// TIA Portal V19 export
FUNCTION "AFC_Steptimer" : Void   // FC35, FBD
TITLE = AFC_Steptimer
{ S7_Optimized_Access := 'TRUE' }
AUTHOR : CH
FAMILY : Aktina
NAME : Global
// AFC_Steptimer
// stored: AutoNumber false, SetENOAutomatically false
   VAR_INPUT
      "step" : Bool;   // Step activated
      count_max : Bool;   // Trigger for max step timer
      count_step : Bool;   // Trigger for conditional step timer
      Pulse : Bool;   // Pulse used for time count
      reset_max : Bool;   // Reset max step timer
      reset_step : Bool;   // Reset conditional step timer
      reset_warn : Bool;   // Reset max timer warning
   END_VAR
   VAR_OUTPUT
      max_warn : Bool;   // Max step timer has elapsed
   END_VAR
   VAR_IN_OUT
      Data : Variant;   // Unique data area for this counter
   END_VAR
   VAR_TEMP
      i : "UDT_STEPTIMER";
      logical1 : Bool;
      remain : UDInt;
      intermediate : UDInt;
      sec : UDInt;
      min : UDInt;
      hour : UDInt;
   END_VAR
BEGIN

REGION Network 1: GEN: Create Logical 1
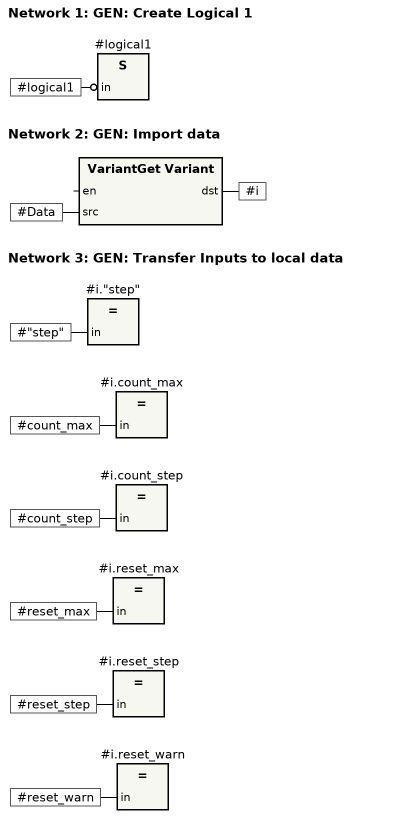
   IF NOT #logical1 THEN #logical1 := TRUE; END_IF;
END_REGION

REGION Network 2: GEN: Import data
   // no SCL statement known for VariantGet: written as a call
   VariantGet(src := #Data, dst => #i);
END_REGION

REGION Network 3: GEN: Transfer Inputs to local data
   #i."step" := #"step";
   #i.count_max := #count_max;
   #i.count_step := #count_step;
   #i.reset_max := #reset_max;
   #i.reset_step := #reset_step;
   #i.reset_warn := #reset_warn;
END_REGION

REGION Network 4: TIMER: Calculate seconds based on h, m, s (max)
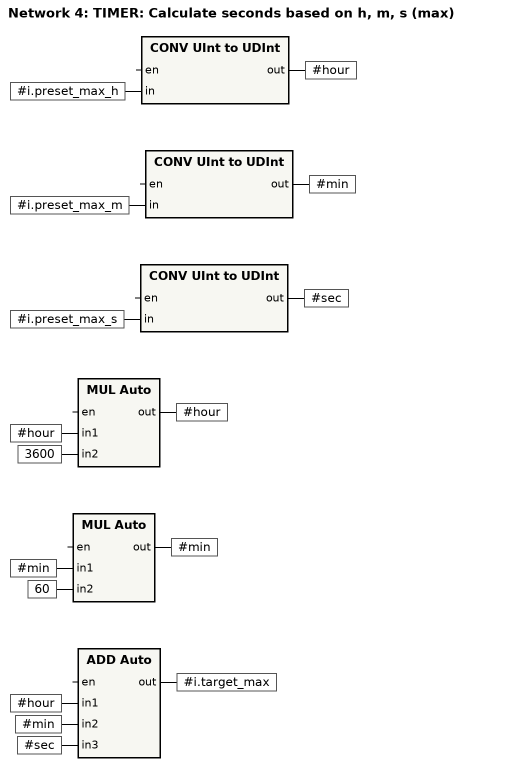
   #hour := UINT_TO_UDINT(#i.preset_max_h);
   #min := UINT_TO_UDINT(#i.preset_max_m);
   #sec := UINT_TO_UDINT(#i.preset_max_s);
   #hour := #hour * 3600;
   #min := #min * 60;
   #i.target_max := #hour + #min + #sec;
END_REGION

REGION Network 5: TIMER: Calculate seconds based on h, m, s (step)
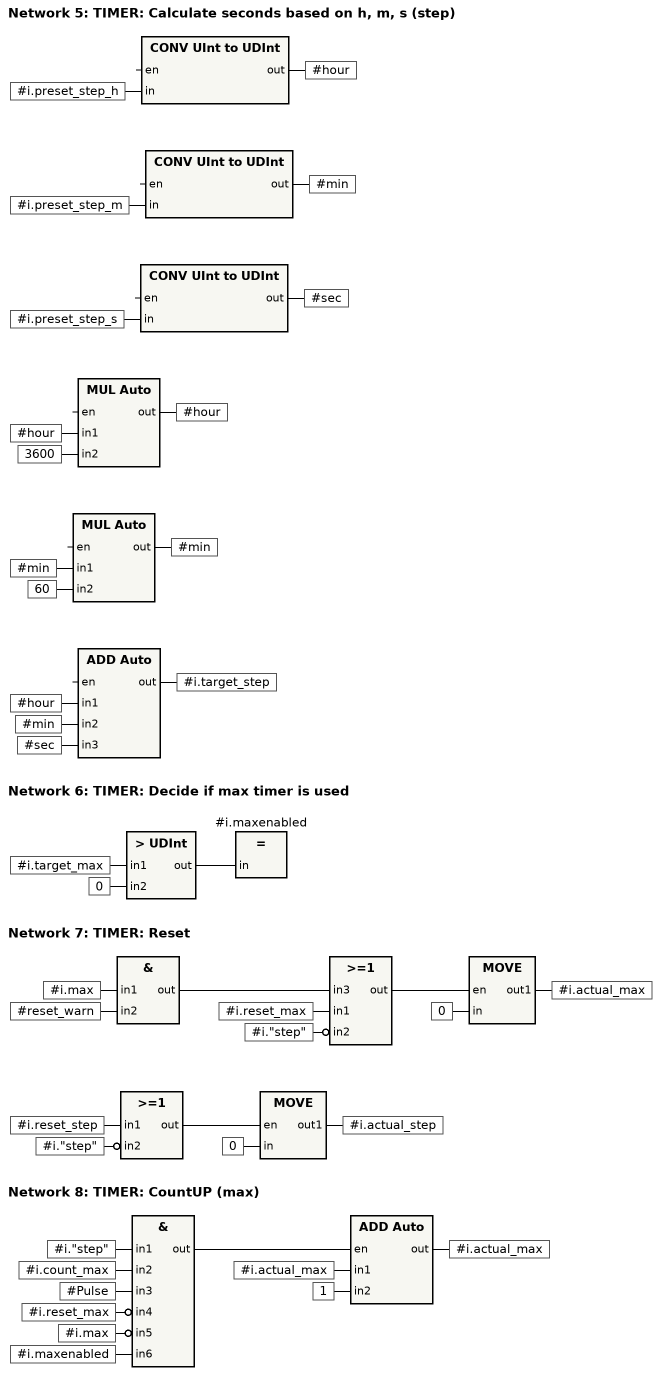
   #hour := UINT_TO_UDINT(#i.preset_step_h);
   #min := UINT_TO_UDINT(#i.preset_step_m);
   #sec := UINT_TO_UDINT(#i.preset_step_s);
   #hour := #hour * 3600;
   #min := #min * 60;
   #i.target_step := #hour + #min + #sec;
END_REGION

REGION Network 6: TIMER: Decide if max timer is used
   #i.maxenabled := #i.target_max > 0;
END_REGION

REGION Network 7: TIMER: Reset
   IF (#i.max AND #reset_warn) OR #i.reset_max OR NOT #i."step" THEN #i.actual_max := 0; END_IF;
   IF #i.reset_step OR NOT #i."step" THEN #i.actual_step := 0; END_IF;
END_REGION

REGION Network 8: TIMER: CountUP (max)
   IF #i."step" AND #i.count_max AND #Pulse AND NOT #i.reset_max AND NOT #i.max AND #i.maxenabled THEN
       #i.actual_max := #i.actual_max + 1;
   END_IF;
END_REGION

REGION Network 9: TIMER: CountUP (step)
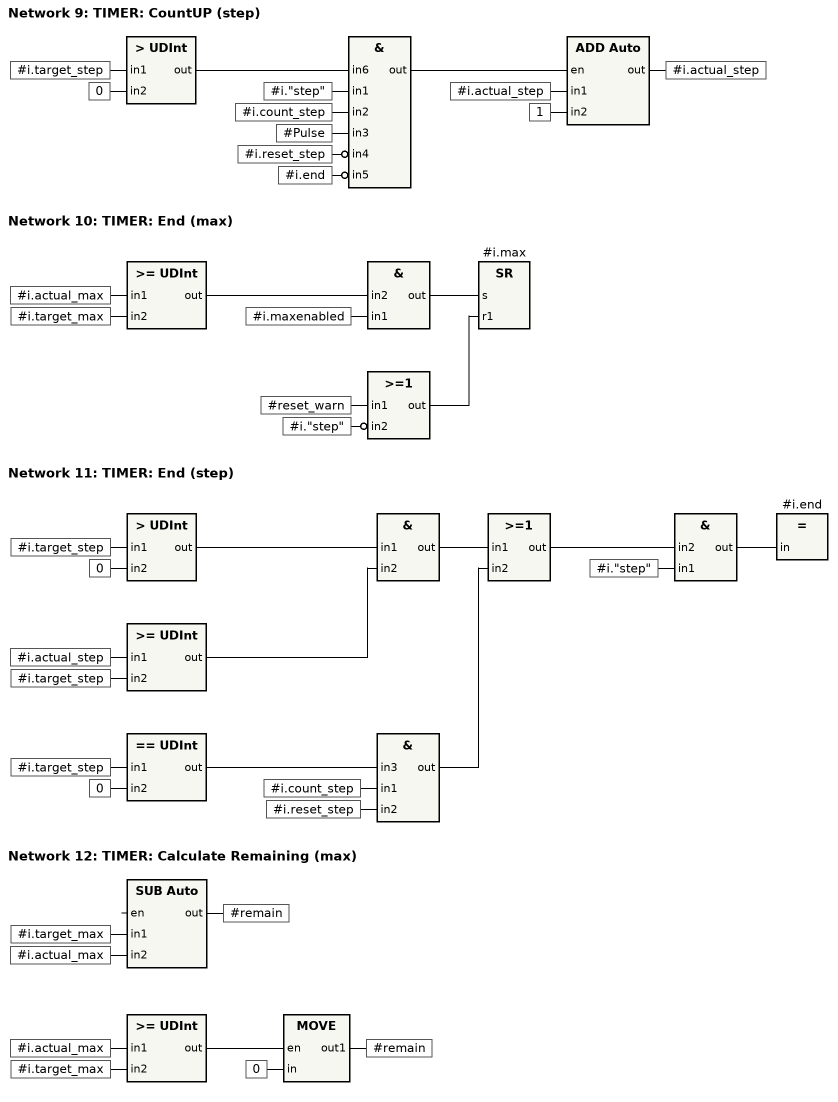
   IF (#i.target_step > 0) AND #i."step" AND #i.count_step AND #Pulse AND NOT #i.reset_step AND NOT #i.end THEN
       #i.actual_step := #i.actual_step + 1;
   END_IF;
END_REGION

REGION Network 10: TIMER: End (max)
   IF (#i.actual_max >= #i.target_max) AND #i.maxenabled THEN
       #i.max := TRUE;   // SR flip-flop
   END_IF;
   IF #reset_warn OR NOT #i."step" THEN #i.max := FALSE; END_IF;
END_REGION

REGION Network 11: TIMER: End (step)
   #i.end := (((#i.target_step > 0) AND (#i.actual_step >= #i.target_step)) OR ((#i.target_step = 0) AND #i.count_step AND #i.reset_step)) AND #i."step";
END_REGION

REGION Network 12: TIMER: Calculate Remaining (max)
   #remain := #i.target_max - #i.actual_max;
   IF #i.actual_max >= #i.target_max THEN #remain := 0; END_IF;
END_REGION

REGION Network 13: TIMER: Convert remaining to h, m, s (max)
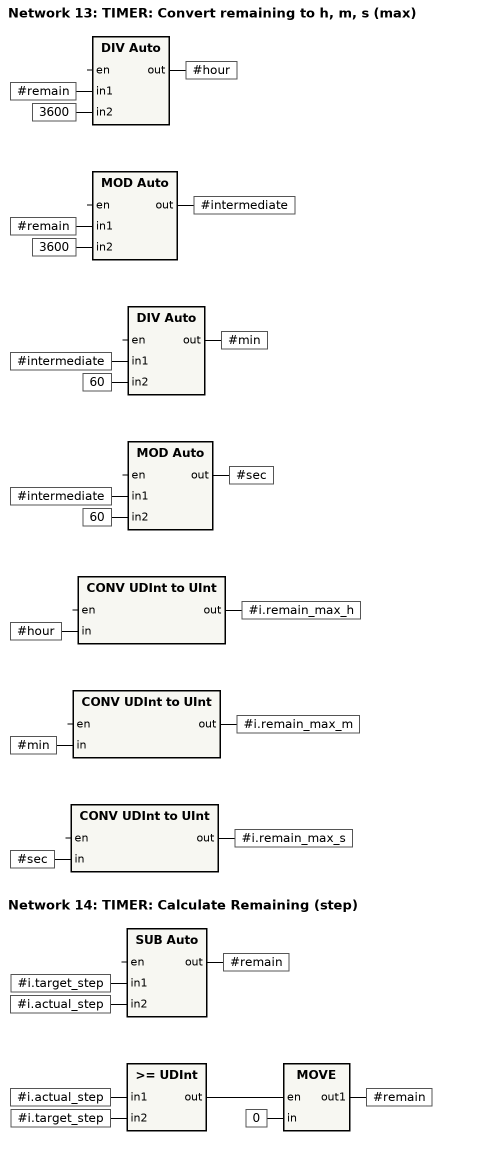
   #hour := #remain / 3600;
   #intermediate := #remain MOD 3600;
   #min := #intermediate / 60;
   #sec := #intermediate MOD 60;
   #i.remain_max_h := UDINT_TO_UINT(#hour);
   #i.remain_max_m := UDINT_TO_UINT(#min);
   #i.remain_max_s := UDINT_TO_UINT(#sec);
END_REGION

REGION Network 14: TIMER: Calculate Remaining (step)
   #remain := #i.target_step - #i.actual_step;
   IF #i.actual_step >= #i.target_step THEN #remain := 0; END_IF;
END_REGION

REGION Network 15: TIMER: Convert remaining to h, m, s (step)
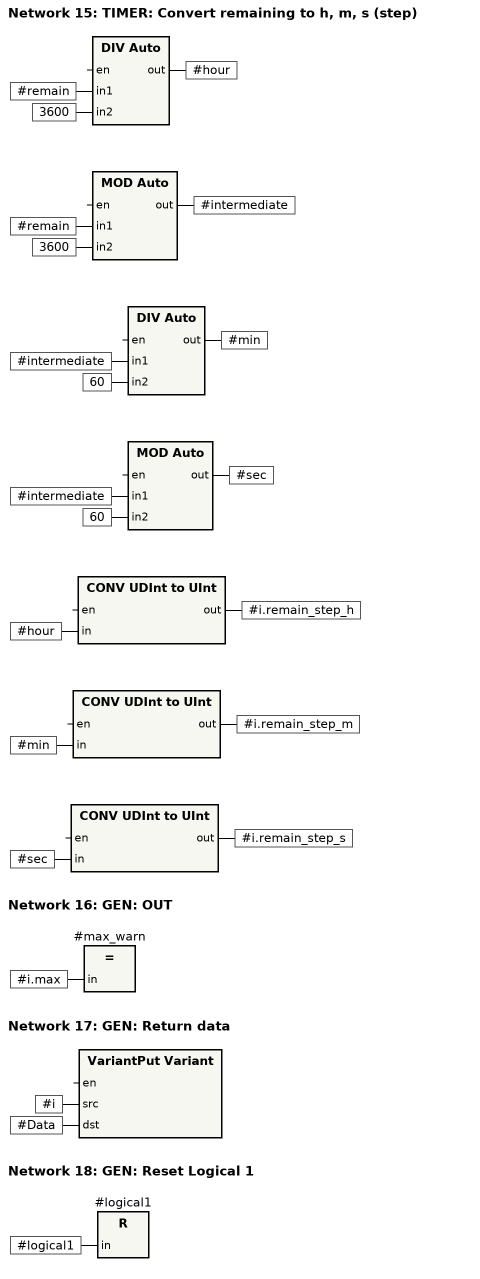
   #hour := #remain / 3600;
   #intermediate := #remain MOD 3600;
   #min := #intermediate / 60;
   #sec := #intermediate MOD 60;
   #i.remain_step_h := UDINT_TO_UINT(#hour);
   #i.remain_step_m := UDINT_TO_UINT(#min);
   #i.remain_step_s := UDINT_TO_UINT(#sec);
END_REGION

REGION Network 16: GEN: OUT
   #max_warn := #i.max;
END_REGION

REGION Network 17: GEN: Return data
   // no SCL statement known for VariantPut: written as a call
   VariantPut(src := #i, dst := #Data);
END_REGION

REGION Network 18: GEN: Reset Logical 1
   IF #logical1 THEN #logical1 := FALSE; END_IF;
END_REGION
END_FUNCTION
